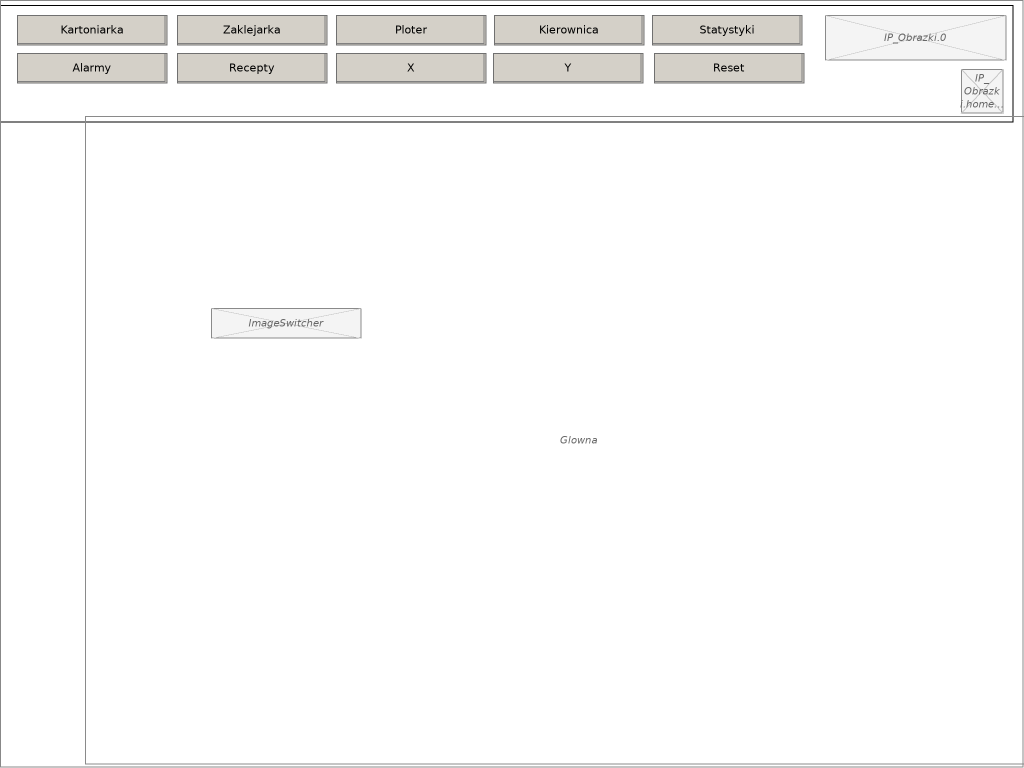
VISUALIZATION HMI  // 1024x768
    Rectangle (-1,5 1014x117)
    Button (17,15 150x30), "Kartoniarka", colour toggle: GVL_HMI.strona=1
        OnMouseDown: FrameSelectionChange Selection=SelectedFrame=f7e3fd18-cbcb-49a2-8593-590d8a027e7f, Selection=1, GlobSel=AssignType=Directly, SelType=Locally
        OnMouseDown: execute { gvl_hmi.strona:=1; }
    Button (177,15 150x30), "Zaklejarka", colour toggle: GVL_HMI.strona=2
        OnMouseDown: FrameSelectionChange Selection=SelectedFrame=f7e3fd18-cbcb-49a2-8593-590d8a027e7f, Selection=7, GlobSel=AssignType=Directly, SelType=Locally
        OnMouseDown: execute { gvl_hmi.strona:=2; }
    Button (654,53 150x30), "Reset", colour toggle: GVL_SafetyFrom_RT2.bSAFETY_PermissionSS1=true and GVL_SafetyFrom_RT2.bSAFETY_PermissionSS2=true
        tap GVL_SafetyFrom_RT2.bSAFETY_ResetCMD
    Button (336,15 150x30), "Ploter", colour toggle: GVL_HMI.strona=3
        OnMouseDown: execute { gvl_hmi.strona:=3; }
        OnMouseDown: FrameSelectionChange Selection=SelectedFrame=f7e3fd18-cbcb-49a2-8593-590d8a027e7f, Selection=3, GlobSel=AssignType=Directly, SelType=Locally
    Button (494,15 150x30), "Kierownica", colour toggle: GVL_HMI.strona=4
        OnMouseDown: execute { gvl_hmi.strona:=4; }
        OnMouseDown: FrameSelectionChange Selection=SelectedFrame=f7e3fd18-cbcb-49a2-8593-590d8a027e7f, Selection=2, GlobSel=AssignType=Directly, SelType=Locally
    Image (825,15 181x45), image: IP_Obrazki.0
    Button (177,53 150x30), "Recepty", colour toggle: GVL_HMI.strona=6
        OnMouseDown: FrameSelectionChange Selection=SelectedFrame=f7e3fd18-cbcb-49a2-8593-590d8a027e7f, Selection=6, GlobSel=AssignType=Directly, SelType=Locally
        OnMouseDown: execute { gvl_hmi.strona:=6; }
    Button (336,53 150x30), "X", colour toggle: GVL_HMI.strona=22
        OnMouseDown: FrameSelectionChange Selection=SelectedFrame=f7e3fd18-cbcb-49a2-8593-590d8a027e7f, Selection=9, GlobSel=AssignType=Directly, SelType=Locally
        OnMouseDown: execute { gvl_hmi.strona:=22; }
    Button (17,53 150x30), "Alarmy", colour toggle: GVL_HMI.strona=5
        OnMouseDown: execute { gvl_hmi.strona:=5; }
        OnMouseDown: FrameSelectionChange Selection=SelectedFrame=f7e3fd18-cbcb-49a2-8593-590d8a027e7f, Selection=8, GlobSel=AssignType=Directly, SelType=Locally
    ImageSwitcher (211,308 150x30), behaviour: TOGGLE
    Image (961,69 42x44), colour toggle: GVL_HMI.strona=0, image: IP_Obrazki.home-icon-silhouette (1)
        OnMouseDown: FrameSelectionChange Selection=SelectedFrame=f7e3fd18-cbcb-49a2-8593-590d8a027e7f, GlobSel=AssignType=Directly, SelType=Locally
        OnMouseDown: execute { gvl_hmi.strona:=0; }
    Button (652,15 150x30), "Statystyki", colour toggle: GVL_HMI.strona=8
        OnMouseDown: execute { gvl_hmi.strona:=8; }
        OnMouseDown: FrameSelectionChange Selection=SelectedFrame=f7e3fd18-cbcb-49a2-8593-590d8a027e7f, Selection=5, GlobSel=AssignType=Directly, SelType=Locally
    Button (493,53 150x30), "Y", colour toggle: GVL_HMI.strona=7
        OnMouseDown: FrameSelectionChange Selection=SelectedFrame=f7e3fd18-cbcb-49a2-8593-590d8a027e7f, Selection=10, GlobSel=AssignType=Directly, SelType=Locally
        OnMouseDown: execute { gvl_hmi.strona:=7; }
    Frame (85,116 988x648)
        shows Glowna()
        shows Kartoniarka()
        shows Kierwonica()
        shows Ploter()
        shows Serwis()
        shows Statystyki()
        shows Visualization()
        shows Zaklejarka()
        shows Alarmy()
        shows PH_AxisOnline(stMcAxisOnline := P_HBot_v3.stMcAxisOnline_MCS_X)
        shows PH_AxisOnline_1(stMcAxisOnline := P_HBot_v3.stMcAxisOnline_MCS_Y)
END_VISUALIZATION

(* stored: Version 1.1.0.1, ProductVersion 3.1.4022.12
   Visu HMI: Id {c5e2f640-41f9-4b33-9695-2524ad6d735c} *)
